// TIA Portal V21 export
FUNCTION_BLOCK "Main GetPut"   // FB6, LAD
{ S7_Optimized_Access := 'TRUE' }
// stored: MemoryReserve 100, SetENOAutomatically false
   VAR
      C { S7_SetPoint := 'True'} : Array[0.."K_NumComunicazioneS7"] of "GestGestPut";
   END_VAR
   VAR_TEMP
      Reset : Bool;
      Update : Bool;
      CounterComunicazione : Int;
      CounterZone : Int;
      Temp_1 : String;
      Temp_2 : String;
   END_VAR
   // // C[1] : QCI
   // // C[2] : Riempitrice
BEGIN

REGION Network 1 (SCL): Reset generale delle comunicazioni
   #Reset := False;
   FOR #CounterZone := 1 TO "K_NumZona" DO
       IF "Zona".Z[#CounterZone].Gen.Reset THEN
           #Reset := True;
       END_IF;
       IF "Zona".Z[#CounterZone].Gen.UpdatePrm THEN
           #Update := True;
       END_IF;
   END_FOR;
   FOR #CounterComunicazione := 0 TO "K_NumComunicazioneS7" DO
       #C[#CounterComunicazione].Reset := #Reset;
       IF #Update THEN
           #C[#CounterComunicazione].K_SegnaleMacchina := 0;
       END_IF;
   END_FOR;
END_REGION

REGION Network 2 (SCL): Comunicazione con QCI
   #C[K_ComunicazioneS7_St1_Qci](Id_Hardware := 16#101,
                                   PuntatoreAreadatiRecivePartner := P#DB9001.DBX0.0 BYTE 208,
                                   PuntatoreAreadatiSendLocale := P#DB9000.dbx0.0  BYTE 208,
                                   PuntatoreAreadatiSendPartner := P#DB9001.DBX208.0 BYTE 204,
                                   PuntatoreAreadatiReciveLocale := P#DB9000.DBX208.0 BYTE 204);
END_REGION

REGION Network 3 (SCL): Comunicazione con ROBOPACK
   #C[K_ComunicazioneS7_St1_Robopack](Id_Hardware := 16#102,
                                        PuntatoreAreadatiRecivePartner := P#DB9001.DBX0.0 BYTE 208,
                                        PuntatoreAreadatiSendLocale := p#DB9000.dbx0.0  BYTE 208,
                                        PuntatoreAreadatiSendPartner := P#DB9001.DBX208.0 BYTE 204,
                                        PuntatoreAreadatiReciveLocale := P#DB9000.DBX208.0 BYTE 204);
END_REGION
END_FUNCTION_BLOCK
